{attribute 'OPC.UA.DA.StructuredType' := '1'}
TYPE ST_TestSystemSetParameters :
STRUCT
	bSystemOperationOn 			: BOOL;
END_STRUCT
END_TYPE

(* stored: Version 1.1.0.1, ProductVersion 3.1.4024.9
   DUT ST_TestSystemSetParameters: Id {6db497b3-3aac-4f76-a37d-b3e8b75b8332} *)
